ORGANIZATION_BLOCK "OB_I_O_Access_Error"
TITLE = %version: 5.06 % %Commit:  % CN: 90
{ S7_Optimized_Access := 'FALSE' }
FAMILY : General
VERSION : 0.0
//Function:
//Module called by CPU when read or write errors occurs
//The operating system calls OB122.
//
//Description:
//The operating system of the CPU calls OB122 whenever
//an error occurs while accessing data on a module. For
//example, if the CPU detects a read error when accessing
//data on an I/O module, the operating system calls OB122.
   VAR_TEMP
      OB122_EV_CLASS : Byte;   // 16#29, Event class 2, Entering event state, Internal fault event
      OB122_SW_FLT : Byte;   // 16#XX Software error code
      OB122_PRIORITY : Byte;   // X = Priority of OB where fault occured (Priority of 1 is lowest)
      OB122_OB_NUMBR : Byte;   // 122 (Organization block 122, OB122)
      OB122_BLK_TYPE : Byte;   // 16#88/8A/8C/8E Type of block fault occured in
      OB122_MEM_AREA : Byte;   // Memory area where access error occured
      OB122_MEM_ADDR : Word;   // Memory address where access error occured
      OB122_BLK_NUM : Word;   // Block number in which error occured
      OB122_PRG_ADDR : Word;   // Program address where error occured
      OB122_DATE_TIME : Date_And_Time;   // Date and time OB1 started
   END_VAR


BEGIN
NETWORK
TITLE = IO Access Error

END_ORGANIZATION_BLOCK

